PROGRAM P_Demo_FB_LicFileGetStorageInfo
VAR
    fbFB_LicFileGetStorageInfo : FB_LicFileGetStorageInfo; // FB_LicFileGetStorageInfo 实例
    bExec                      : BOOL := FALSE;
    bBusy_                     : BOOL;
    bErrFlag                   : BOOL;
    nErrCode                   : UDINT;
END_VAR

// =============================================================================
// 场景：查 dongle 存储。
// 价值：预检支持。
// 验证：触发后观察 bDone / bErr，错误号 nErrId 反映 ADS Return Codes。
// 验证步骤：
//   1. 右键 PLC 项目下 POUs 文件夹 → Add → Existing Item → 选本 .TcPOU 文件
//   2. 引用 Tc2_Utilities（References → Add library）
//   3. 编译 → 登录 → 运行；按上方『验证』行的指示在线写值观察
// =============================================================================

fbFB_LicFileGetStorageInfo(
    bExecute := bExec, tTimeout := DEFAULT_ADS_TIMEOUT,
    bBusy => bBusy_, bError => bErrFlag, nErrorId => nErrCode
);

END_PROGRAM

(* stored: Version 1.1.0.1, ProductVersion 3.1.4024.5
   POU P_Demo_FB_LicFileGetStorageInfo: Id {b57ad1e9-43b8-5681-9a43-3460569a2a5e}, SpecialFunc None *)
